SUBAPPLICATION LD_helper (* Subapplication Type *)
  (* Standard: 61499-2 *)
  (* Version 1.0, 2026-05-04, franz *)
  PACKAGE FBs::Counter::subs::Zaehler;
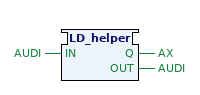
  SOCKETS
    IN : adapter::types::unidirectional::AUDI;
  END_SOCKETS
  PLUGS
    Q : adapter::types::unidirectional::AX;
    OUT : adapter::types::unidirectional::AUDI;
  END_PLUGS
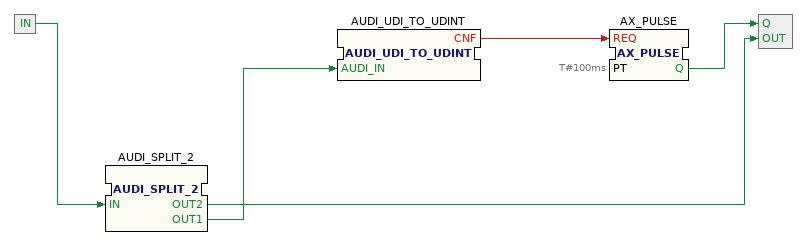
  FBS
    AX_PULSE : adapter::events::unidirectional::timers::AX_PULSE(PT := T#100ms);
    AUDI_SPLIT_2 : adapter::events::unidirectional::AUDI_SPLIT_2;
    AUDI_UDI_TO_UDINT : adapter::conversion::unidirectional::AUDI_UDI_TO_UDINT;
  END_FBS
  EVENT_CONNECTIONS
    AUDI_UDI_TO_UDINT.CNF TO AX_PULSE.REQ;
  END_CONNECTIONS
  ADAPTER_CONNECTIONS
    IN TO AUDI_SPLIT_2.IN;
    AUDI_SPLIT_2.OUT2 TO OUT;
    AX_PULSE.Q TO Q;
    AUDI_SPLIT_2.OUT1 TO AUDI_UDI_TO_UDINT.AUDI_IN;
  END_CONNECTIONS
END_SUBAPPLICATION
